// TIA Portal V17 export
// export: Created 2022-12-09T10:51:18.0947432Z, ExportSetting WithDefaults, DisplayName Totally Integrated Automation Portal, DisplayVersion V17 Update 5, DisplayName TIA Portal Openness, DisplayVersion V17 Update 5, DisplayName TIA Portal Version Control Interface, DisplayVersion V17, DisplayName Simotion SCOUT TIA, DisplayVersion 5.4.3.0, DisplayName SINAMICS Startdrive Advanced, DisplayVersion V17 SP1, DisplayName SINAMICS Startdrive G130, G150, S120, S150, SINAMICS MV, S210, DisplayVersion V17 SP1, DisplayName SINAMICS Startdrive G110M, G120, G120C, G120D, G120P, G115D, DisplayVersion V17 SP1, DisplayName STEP 7 Professional, DisplayVersion V17 Update 5, DisplayName STEP 7 Safety, DisplayVersion V17, DisplayName WinCC Advanced, DisplayVersion V17 Update 5
TYPE "UDT_SIKOPARAMETER"
// stored: IsFailsafeCompliant false
   STRUCT
      DecimalPlaces : Byte;   // 0 - 1; 1 - 0.1; 2 - 0.01; 3 - 0.001
      DirectionIndicators : Byte;   // 0 - cw; 1 - ccw
      DisplayOrientation : Byte;   // 0 - 0°; 1 - 180°
      CountingDirection : Byte;   // 0 - cw; 1 - ccw
      ResolutionPerRevolution : Int;   // 20 - ; 25 - ; 40 - ; 80 - ;
      OffsetValue : Int;
      CalibrationValue : DInt;
      TargetWindow1 : Int;
      PositioningType : Byte;
      LoopLength : Int;
      OperatingMode : Byte;
   END_STRUCT;
END_TYPE
